FUNCTION_BLOCK Time_Count (* Basic Function Block Type *)
  (* Standard: 61499-2 *)
  (* Version 0.0, 7/6/2016, gulzha, nxtControl GmbH, Template *)
  PACKAGE Main;
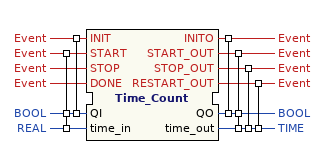
  EVENT_INPUT
    INIT WITH QI; (* Initialization Request *)
    START WITH QI, time_in; (* Normal Execution Request *)
    STOP;
    DONE;
  END_EVENT
  EVENT_OUTPUT
    INITO WITH QO; (* Initialization Confirm *)
    START_OUT WITH QO, time_out; (* Execution Confirmation *)
    STOP_OUT WITH time_out;
    RESTART_OUT WITH time_out;
  END_EVENT
  VAR_INPUT
    QI : BOOL; (* Input event qualifier *)
    time_in : REAL;
  END_VAR
  VAR_OUTPUT
    QO : BOOL; (* Output event qualifier *)
    time_out : TIME;
  END_VAR
  VAR
    TimeStampStart : DATE_AND_TIME;
    TimeStampRestart : DATE_AND_TIME;
    time_elapsed : TIME := 0;
    started : BOOL := FALSE;
    time_in_internal : TIME;
  END_VAR
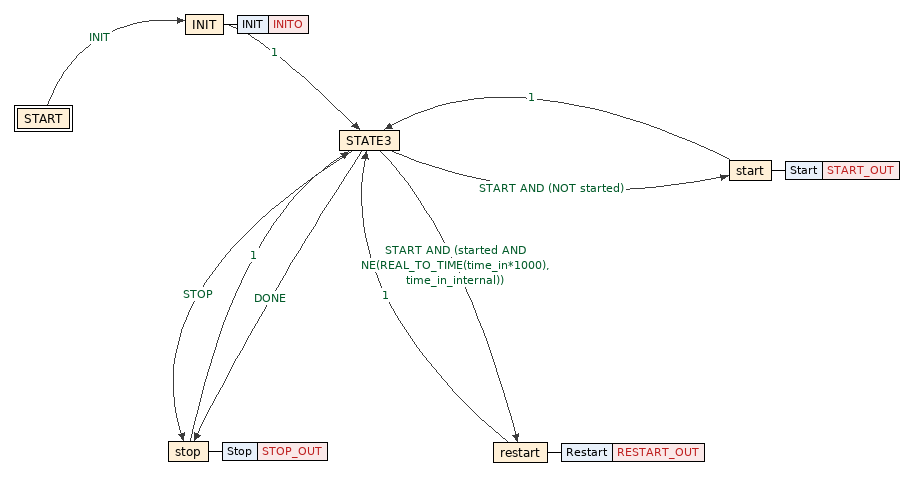
  EC_STATES
    START; (* Initial State *)
    INIT : INIT -> INITO; (* Initialization *)
    start : Start -> START_OUT; (* Normal execution *)
    restart : Restart -> RESTART_OUT;
    stop : Stop -> STOP_OUT;
    STATE3;
  END_STATES
  EC_TRANSITIONS
    START TO INIT := INIT;
    INIT TO STATE3 := 1;
    restart TO STATE3 := 1;
    STATE3 TO stop := DONE;
    STATE3 TO stop := STOP;
    stop TO STATE3 := 1;
    start TO STATE3 := 1;
    STATE3 TO start := START AND (NOT started);
    STATE3 TO restart := START AND (started AND NE(REAL_TO_TIME(time_in*1000), time_in_internal));
  END_TRANSITIONS
  ALGORITHM INIT IN ST: (* Initialization algorithm *)
;
//time_out:=0;
//time_elapsed:=0;
//TimeStampRestart := 0;
//TimeStampStart := 0;
started := FALSE;
//time_in_internal := 0;
  END_ALGORITHM
  ALGORITHM Start IN ST: (* Normally executed algorithm *)
;

TimeStampStart := CURRENT_DT();
time_in_internal := REAL_TO_TIME(time_in*1000);
time_out := time_in_internal;
started := TRUE;

//time_out := REAL_TO_TIME(time_in*1000); // convert seconds into ms, then convert it into TIME format
  END_ALGORITHM
  ALGORITHM Restart IN ST:
;

TimeStampRestart := CURRENT_DT();
time_in_internal := REAL_TO_TIME(time_in*1000);

time_elapsed := SUB_DT_DT(TimeStampRestart, TimeStampStart);
//time_elapsed := D TimeStampRestart - TimeStampStart;
time_out := time_in_internal- time_elapsed;
  END_ALGORITHM
  ALGORITHM Stop IN ST:
;


//time_out:=0;
//time_elapsed:=0;
//TimeStampRestart := 0;
//TimeStampStart := 0;
started := FALSE;
  END_ALGORITHM
END_FUNCTION_BLOCK
